// TIA Portal V19 export
DATA_BLOCK "P_TRIG"   // DB21
{ S7_Optimized_Access := 'TRUE' }
// stored: MemoryReserve 100
   VAR
      ARR : Array[0..100] of Bool;
   END_VAR
BEGIN
END_DATA_BLOCK
